(****************************************************************
NAME:			FB_SetAxisPosition
DATA:			2017.2.16
VERSION:		1.0.0
DESCRIPTION:	FB_SetAxisPosition
HISTORY:
				2017.2.16		NEW

***************************************************************)
FUNCTION_BLOCK FB_SetAxisPosition
VAR_INPUT
	//GapValueSet:LREAL:=0;
	ValueSet_PhaseShifterLin:LREAL:=0;
	Execute:BOOL;
END_VAR
VAR_OUTPUT
	FbID:DINT:=1001;
	State:DINT;
	Busy:BOOL;
	Done:BOOL;
	Error:BOOL;
	ErrorID:DINT;
END_VAR
VAR
	PhaseShifterLin_MC_SetPosition: MC_SetPosition;
	fb_ton: TON;
	FB_PlcEmergencyStop: FB_PlcEmergencyStop;
END_VAR

IF Execute THEN
Busy:=TRUE;
Done:=FALSE;
fb_ton(PT:=t#0.1s);
CASE State OF
	0:
		IF PhaseShifterLin_MC_SetPosition.Error  THEN		(*FB Error*)
			ErrorID:=1;
			State:=99;
		END_IF
		State:=1;
	1:	(*Execute*)
		PhaseShifterLin_MC_SetPosition.Position:=ValueSet_PhaseShifterLin;
		PhaseShifterLin_MC_SetPosition.Execute:=TRUE;
		A_SetPositionMC();
		fb_ton.IN:=TRUE;
		State:=2;
	2:	(*Wait*)
		A_SetPositionMC();
		IF NOT PhaseShifterLin_MC_SetPosition.Done THEN		(*DoneÐÅºÅ²»µ½£¬¼ÌÐøµÈ´ý£¬Èç¹û³¬Ê±ÔòFB Error*)
			IF NOT fb_ton.Q THEN
				State:=2;
			ELSE
				ErrorID:=4;
				State:=99;
			END_IF
		ELSIF  PhaseShifterLin_MC_SetPosition.Done THEN		(*Done£¬×ªÏÂÒ»²½*)
			State:=88;
		ELSE
			ErrorID:=5;
			State:=99;
		END_IF
	88:
		Execute:=FALSE;
		State:=0;
		Busy:=FALSE;
		Done:=TRUE;
		Error:=FALSE;
		ErrorID:=0;
		PhaseShifterLin_MC_SetPosition.Execute:=FALSE;
		fb_ton.IN:=FALSE;
	99:
		Execute:=FALSE;
		State:=99;
		Busy:=FALSE;
		Done:=FALSE;
		Error:=TRUE;
		PhaseShifterLin_MC_SetPosition.Execute:=FALSE;
		fb_ton.IN:=FALSE;
	-100:
		FB_PlcEmergencyStop();
		Execute:=FALSE;
		State:=-100;
		Busy:=FALSE;
		Done:=FALSE;
		Error:=TRUE;
		PhaseShifterLin_MC_SetPosition.Execute:=FALSE;
		fb_ton.IN:=FALSE;
END_CASE
END_IF

ACTION A_SetPositionMC:
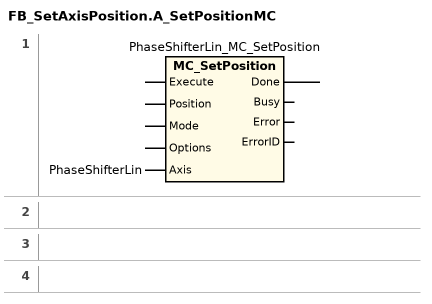
// NETWORK 1
PhaseShifterLin_MC_SetPosition(Axis := PhaseShifterLin); // MC_SetPosition

// NETWORK 2

// NETWORK 3

// NETWORK 4
END_ACTION

END_FUNCTION_BLOCK

(* stored: Version 1.1.0.1, ProductVersion 3.1.4024.6
   POU FB_SetAxisPosition: Id {6afa31ff-e0ae-4621-979a-f7f274bb3d8a}, SpecialFunc None
   Action A_SetPositionMC: Id {9afeaa97-7af6-44a0-91c2-9bb3ac449bed} *)
